Yaskawa INFORM job: MULTI-ABOVE.JBI

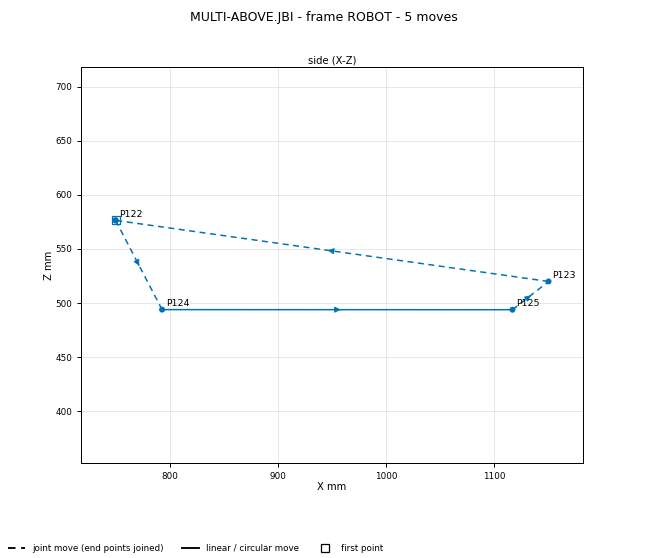
[picture p0: tool path of MULTI-ABOVE.JBI in frame ROBOT, 5 of 5 moves have a stored position in this frame; points joined in program order, loops and branches not executed]
/JOB
//NAME MULTI-ABOVE
///FOLDERNAME FOLDER001
//POS
///NPOS 2,0,0,4,0,0
///USER 15
///TOOL 1
///POSTYPE USER
///RECTAN
///RCONF 1,0,0,0,0,0,0,0,0,0,0,0,0,0,0,0,0,0,0,0,0,0,0,0
C00000=4.666,-1.318,179.409,180.0000,-10.0000,0.0000
C00001=4.513,-65.064,179.402,180.0000,-10.0000,0.0000
///POSTYPE ROBOT
P00122=750.004,162.000,576.437,180.0000,-9.9968,0.0000
P00123=1150.002,160.000,520.003,180.0000,-25.0002,0.0000
P00124=792.896,161.791,493.972,179.9986,-9.9993,0.0008
P00125=1116.664,160.780,493.887,-179.9993,-9.9981,-0.0025
//INST
///DATE 2025/05/27 07:28
///ATTR SC,RW,RJ
////FRAME USER 15
///GROUP1 RB1
///LVARS 20,20,20,0,0,0,0,0
NOP
GETARG LB000 IARG#(1)
ADD B096 LB000
'=========
DOUT OT#(46) ON
TIMER T=0.50
JUMP LABEL: B098
*0
'ROOT
SFTOF
MACRO1 MJ#(2) ARGF2.4 ARGF1.5 ARGF0.0
MACRO1 MJ#(1) ARGF0.0 ARGF0.0 ARGF0.0 ARGF0.0 ARGF0.0 ARGF0.0
JUMP *LABEL
*1
'LAYER 1 - 1
SFTOF
MACRO1 MJ#(2) ARGF0.5 ARGF1.0 ARGF0.0
MACRO1 MJ#(1) ARGF0.0 ARGF-1.5 ARGF3.0 ARGF-5.0 ARGF0.0 ARGF0.0
JUMP *LABEL
*2
'LAYER 1 - 2
SFTOF
MACRO1 MJ#(2) ARGF0.5 ARGF1.0 ARGF0.0
MACRO1 MJ#(1) ARGF0.0 ARGF1.5 ARGF3.0 ARGF5.0 ARGF0.0 ARGF0.0
JUMP *LABEL
*3
'LAYER 2 - 1
SFTOF
MACRO1 MJ#(2) ARGF0.5 ARGF1.0 ARGF0.0
MACRO1 MJ#(1) ARGF0.0 ARGF3.0 ARGF6.0 ARGF7.0 ARGF0.0 ARGF0.0
JUMP *LABEL
*4
'LAYER 2 -2
SFTOF
MACRO1 MJ#(2) ARGF0.5 ARGF1.0 ARGF0.0
MACRO1 MJ#(1) ARGF0.0 ARGF-3.0 ARGF6.0 ARGF-7.0 ARGF0.0 ARGF0.0
JUMP *LABEL
*5
'LAYER 3 - 1
SFTOF
MACRO1 MJ#(2) ARGF0.5 ARGF1.0 ARGF0.0
MACRO1 MJ#(1) ARGF0.0 ARGF-6.0 ARGF9.0 ARGF-7.0 ARGF0.0 ARGF0.0
JUMP *LABEL
*6
'LAYER 3 - 2
SFTOF
MACRO1 MJ#(2) ARGF0.5 ARGF1.0 ARGF0.0
MACRO1 MJ#(1) ARGF0.0 ARGF0.0 ARGF9.0 ARGF0.0 ARGF0.0 ARGF0.0
JUMP *LABEL
*7
'LAYER 3 - 3
SFTOF
MACRO1 MJ#(2) ARGF0.5 ARGF1.0 ARGF0.0
MACRO1 MJ#(1) ARGF0.0 ARGF6.0 ARGF9.0 ARGF7.0 ARGF0.0 ARGF0.0
JUMP *LABEL
*8
'LAYER 4 - 1
SFTOF
MACRO1 MJ#(2) ARGF0.5 ARGF1.0 ARGF0.0
MACRO1 MJ#(1) ARGF0.0 ARGF9.0 ARGF13.0 ARGF7.0 ARGF0.0 ARGF0.0
JUMP *LABEL
*9
'LAYER 4 - 2
SFTOF
MACRO1 MJ#(2) ARGF0.5 ARGF1.0 ARGF0.0
MACRO1 MJ#(1) ARGF0.0 ARGF3.0 ARGF13.0 ARGF0.0 ARGF0.0 ARGF0.0
JUMP *LABEL
*10
'LAYER 4 - 3
SFTOF
MACRO1 MJ#(2) ARGF0.5 ARGF1.0 ARGF0.0
MACRO1 MJ#(1) ARGF0.0 ARGF-9.0 ARGF13.0 ARGF-7.0 ARGF0.0 ARGF0.0
JUMP *LABEL
*11
'LAYER 4 - 4
SFTOF
MACRO1 MJ#(2) ARGF0.5 ARGF1.0 ARGF0.0
MACRO1 MJ#(1) ARGF0.0 ARGF-3.0 ARGF13.0 ARGF-7.0 ARGF0.0 ARGF0.0
JUMP *LABEL
*12
'LAYER 5 - 1
SFTOF
MACRO1 MJ#(2) ARGF0.5 ARGF1.0 ARGF0.0
MACRO1 MJ#(1) ARGF0.0 ARGF12.0 ARGF18.0 ARGF7.0 ARGF0.0 ARGF0.0
JUMP *LABEL
*13
'LAYER 5 - 2
SFTOF
MACRO1 MJ#(2) ARGF0.5 ARGF1.0 ARGF0.0
MACRO1 MJ#(1) ARGF0.0 ARGF6.0 ARGF18.0 ARGF0.0 ARGF0.0 ARGF0.0
JUMP *LABEL
*14
'LAYER 5 - 3
SFTOF
MACRO1 MJ#(2) ARGF0.5 ARGF1.0 ARGF0.0
MACRO1 MJ#(1) ARGF0.0 ARGF12.0 ARGF18.0 ARGF7.0 ARGF0.0 ARGF0.0
JUMP *LABEL
*15
'LAYER 5 - 4
SFTOF
MACRO1 MJ#(2) ARGF0.5 ARGF1.0 ARGF0.0
MACRO1 MJ#(1) ARGF0.0 ARGF-6.0 ARGF18.0 ARGF0.0 ARGF0.0 ARGF0.0
JUMP *LABEL
*16
'LAYER 5 - 5
SFTOF
MACRO1 MJ#(2) ARGF0.5 ARGF1.0 ARGF0.0
MACRO1 MJ#(1) ARGF0.0 ARGF0.0 ARGF18.0 ARGF0.0 ARGF0.0 ARGF0.0
JUMP *LABEL
*LABEL
REFP 1 C00000
REFP 2 C00001
MOVJ P122 VJ=15.00 PL=3
MOVJ P124 VJ=15.00 PL=0
ARCON
WVON AMP=D080 FREQ=D081 ANGL=D082
MOVL P125 V=25.0 PL=0
WVOF
ARCOF
MOVJ P123 VJ=15.00 PL=3
MOVJ P122 VJ=15.00 PL=3
INC B098
SFTOF
JUMP LABEL: B098 IF B098<B096
SET B098 B096
END
